{attribute 'linkalways'} 
{attribute 'no_explicit_call' := 'This FB is a CLASS and must be accessed using methods or properties'}
{attribute 'enable_dynamic_creation'}
FUNCTION_BLOCK Node_F_VN_SetAt_TcVnRectangle_DINT EXTENDS VisionNode
VAR
    stElement : _TcVnRectangle_DINT;
    ipContainer : _ITcVnContainer;
    nIndex : _ULINT(0);
    hrPrev : _HRESULT(S_OK);
    hresult : _HRESULT(S_OK);
END_VAR

METHOD PUBLIC  Clone : I_Node
VAR
	pNode : POINTER TO Node_F_VN_SetAt_TcVnRectangle_DINT;
END_VAR
pNode := __NEW(Node_F_VN_SetAt_TcVnRectangle_DINT);
Clone := pNode^;
END_METHOD

METHOD FB_init : BOOL
VAR_INPUT
	bInitRetains : BOOL; // if TRUE, the retain variables are initialized (warm start / cold start)
	bInCopyCode : BOOL;  // if TRUE, the instance afterwards gets moved into the copy code (online change)
END_VAR
AddInput('stElement', stElement);
AddInput('ipContainer', ipContainer);
AddInput('nIndex', nIndex);
AddInput('hrPrev', hrPrev);
AddOutput('ipContainer', ipContainer);
AddOutput('hresult',hresult);
END_METHOD

METHOD PROTECTED OnExecute : HRESULT
hresult.Value := F_VN_SetAt_TcVnRectangle_DINT(
    stElement := stElement.Value,
    ipContainer := ipContainer.Value,
    nIndex := nIndex.Value,
    hrPrev:= hrPrev.Value);
END_METHOD

METHOD PUBLIC PreExecutionCheck
VAR_INPUT
	Check : I_PreExecutionChecks;
END_VAR
Check.IsTrue(ipContainer.IsValid, 'ipContainer must be a valid container');
END_METHOD

END_FUNCTION_BLOCK

(* stored: Version 1.1.0.1, ProductVersion 3.1.4024.13
   POU Node_F_VN_SetAt_TcVnRectangle_DINT: Id {65cb1eed-6bd1-4108-8ad8-673a714b427d}, SpecialFunc None
   Folder Constructor: Id {4827cc74-1668-4f46-8777-35857cd9c312}
   Method Clone: Id {3670f4da-e911-46c1-abe7-f5bd962ea87e}
   Method FB_init: Id {125d5c18-a970-45dd-9374-2d7807333f88}
   Method OnExecute: Id {528cc1d1-0e8f-4dd7-9c06-cf08f535705d}
   Method PreExecutionCheck: Id {121ff92e-d9d9-4519-b624-b6f4121a5798} *)
